TYPE VoltageRegulation_Struct :
UNION
		Value : INT;
		Bits : Bits_VoltageRegulation;
END_UNION
END_TYPE

(* stored: Version 1.1.0.1, ProductVersion 3.1.4022.18
   DUT VoltageRegulation_Struct: Id {9843a29b-146e-48d0-89c9-13651ddd8309} *)
